TYPE ST_OverloadAL :
STRUCT
	Status:	BIT;
END_STRUCT
END_TYPE

(* stored: Version 1.1.0.1, ProductVersion 3.1.4020.6
   DUT ST_OverloadAL: Id {cdc893ac-6fb2-4fda-aa0d-53b1711d4396} *)
